// TIA Portal V17 export
// export: Created 2024-09-03T21:54:56.5708123Z, ExportSetting WithDefaults, DisplayName Totally Integrated Automation Portal, DisplayVersion V17 Update 7, DisplayName TIA Portal Openness, DisplayVersion V17 Update 7, DisplayName TIA Portal Version Control Interface, DisplayVersion V17, DisplayName SINAMICS Startdrive Advanced, DisplayVersion V17 SP2, DisplayName SINAMICS Startdrive G110M, G120, G120C, G120D, G120P, G115D, DisplayVersion V17 SP2, DisplayName SINAMICS Startdrive G130, G150, S120, S150, SINAMICS MV, S210, DisplayVersion V17 SP2, DisplayName STEP 7 Professional, DisplayVersion V17 Update 7, DisplayName STEP 7 Safety, DisplayVersion V17 Update 6, DisplayName WinCC Advanced / Unified PC, DisplayVersion V17 Update 7
DATA_BLOCK "AutoPositions"   // DB11
{ S7_Optimized_Access := 'TRUE' }
VERSION : 0.1
// stored: AutoNumber true, DBAccessibleFromOPCUA true, DBAccessibleFromWebserver true, IsOnlyStoredInLoadMemory false, IsRetainMemResEnabled false, IsWriteProtectedInAS false, MemoryReserve 100
   VAR RETAIN
      St1_Table1 : "UDT_PositionData";
      St2_Table2 : "UDT_PositionData";
      St3_Fitting : "UDT_PositionData";
      R1_Gripper : "UDT_PositionData";
      AE_Gripper : "UDT_PositionData";
      St4_OKposition : "UDT_PositionData";
   END_VAR
   VAR
      emptyPos : "UDT_PositionData";
   END_VAR
BEGIN
END_DATA_BLOCK
